FUNCTION_BLOCK ExecuteManual EXTENDS Vanguard_WaferDetection.State
VAR
	_stateMachine : I_ExecuteTranisitons;
	ChannelControl : I_VisionChannelControl;
	OperatingState : INT;
	DummySKUDetectedSignal : BOOL;
	startTrig : R_TRIG;
	stopTrig : R_TRIG;
	skuTrigger : R_TRIG;
END_VAR

METHOD Executing : BOOL
skuTrigger(CLK := DummySKUDetectedSignal);
CASE OperatingState OF 
	0:
		IF skuTrigger.Q THEN
			ChannelControl.TriggerImage();
			OperatingState := 1;
		END_IF
	1:
		IF ChannelControl.ImageProcessing THEN
			OperatingState := 2;
		END_IF
	2:
		IF ChannelControl.ImageProcessingCompletedSuccessfully THEN
			OperatingState := 0;
		ELSE
			OperatingState := 99;
		END_IF
END_CASE
END_METHOD

//FB_Init is always available implicitly and it is used primarily for initialization.
//The return value is not evaluated. For a specific influence, you can also declare the
//methods explicitly and provide additional code there with the standard initialization
//code. You can evaluate the return value.
METHOD FB_Init: BOOL
VAR_INPUT
    bInitRetains: BOOL; // TRUE: the retain variables are initialized (reset warm / reset cold)
    bInCopyCode: BOOL;  // TRUE: the instance will be copied to the copy code afterward (online change)   
	StateMachine : I_ExecuteTranisitons;
END_VAR
_stateMachine := StateMachine;
END_METHOD

METHOD SetDependencies : BOOL
VAR_INPUT
	Control : I_VisionChannelControl;
END_VAR
ChannelControl := Control;
END_METHOD

END_FUNCTION_BLOCK

(* stored: Version 1.1.0.1
   POU ExecuteManual: Id {532a6e25-2d18-498d-b6ba-e63eba45ba25}, SpecialFunc None
   Method Executing: Id {d30b50e2-6397-41cc-aca9-1c7af7d8bf62}
   Method FB_Init: Id {a811cb79-0054-4aea-8c66-80334a792822}
   Method SetDependencies: Id {d669ca64-0d81-4293-83f8-fc69f95a029d} *)
